(* IEC 61131-3 sources: generating_plc_code_with_llms/Code#2/CodeLlama/first run, 21 files *)

(* ---- 10.st ---- *)
// 23.71102786064148s
// 2
```
FUNCTION SIGMOID(X:REAL):REAL
VAR
    Y:REAL;
END_VAR
IF (X>0) THEN
    Y:=1/(1+EXP(-X));
ELSE
    Y:=1-1/(1+EXP(X));
END_IF;
RETURN Y;
END_FUNCTION;
```

(* ---- 11.st ---- *)
// 28.231884717941284s
// 2
```
FUNCTION sign(x : REAL) : REAL;
VAR
    y : REAL;
END_VAR
IF (x > 0.0) THEN
    y := 1.0;
ELSIF (x < 0.0) THEN
    y := -1.0;
ELSE
    y := 0.0;
END_IF
RETURN y;
END_FUNCTION
```

(* ---- 12.st ---- *)
// 19.33155584335327s
// 2
```
FUNCTION SINH(X:REAL):REAL;
BEGIN
    RETURN EXP(X) - 1/EXP(X);
END_FUNCTION;
```

(* ---- 13.st ---- *)
// 41.79835319519043s
// 2
```
FUNCTION SelectNumber(nNumber : INT) : BOOL;
VAR
    bFound : BOOL := FALSE;
END_VAR

bFound := FALSE;
REPEAT
    IF aNumbers[nCnt] = nNumber THEN
        bFound := TRUE;
        EXIT;
    END_IF;
    nCnt := nCnt + 1;
UNTIL (nCnt > MAXNUMBERS) OR (bFound);

IF NOT(bFound) AND (aNumbers[nCnt] = 10) THEN
    EXIT;
END_IF;

RETURN bFound;
END_FUNCTION;
```

(* ---- 14.st ---- *)
// 54.95126724243164s
// 3
```
FUNCTION FC1001 :BOOL
VAR_INPUT
	MEW: REAL;
	SP: REAL;
	HYS: REAL;
END_VAR
VAR_IN_OUT
 	OUT:BOOL;
END_VAR
VAR
 	P_HYS: REAL;
END_VAR
BEGIN
  IF (MEW > SP) THEN
    P_HYS := HYS / 100 * SP;
    IF (MEW - P_HYS > 0) THEN
      OUT := TRUE;
    ELSE
      OUT := FALSE;
    END_IF;
  ELSE
    P_HYS := HYS / 100 * MEW;
    IF (P_HYS - SP > 0) THEN
      OUT := TRUE;
    ELSE
      OUT := FALSE;
    END_IF;
  END_IF;
END_FUNCTION
```

(* ---- 15.st ---- *)
// 47.454710721969604s
// 2
```
FUNCTION FC1002 :BOOL
VAR_INPUT
	E_A, SENSOR: BOOL;
	ZEITW: TIME;
END_VAR
VAR_IN_OUT
	ZEIT:TON;
	P_HU, P_AL: BOOL;
END_VAR
BEGIN
	IF E_A THEN
		IF SENSOR THEN
			P_HU := TRUE;
			ZEIT := ZEITW;
		ELSE
			IF (ZEITW - ZEIT) > T#3s THEN
				P_AL := TRUE;
			END_IF;
		END_IF;
	END_IF;
END_FUNCTION;
```

(* ---- 17.st ---- *)
// 48.49951720237732s
// 2
```
FUNCTION TEXT_OUTPUT
VAR
    iTemp : INT;
    iHumidity : INT;
END_VAR
iTemp := aiOutside;
iHumidity := aiHumidity;
IF (iTemp < 18) THEN
    sShowText := "Cold";
ELSIF (iTemp >= 18 AND iTemp <= 25) THEN
    IF (iHumidity >= 40 AND iHumidity <= 75) THEN
        sShowText := "Opt";
    ELSE
        sShowText := "Temp. OK";
    END_IF;
ELSE
    sShowText := "Hot";
END_IF;
sShowText;
END_FUNCTION;
```

(* ---- 18.st ---- *)
// 54.627214670181274s
// 4

```
FUNCTION FC1003 : VOID
VAR_INPUT
    IN_R:REAL;
    IN_MAX, IN_MIN:REAL;
    OUT_MAX, OUT_MIN:REAL;
END_VAR
VAR_OUTPUT
    OUT_R:REAL;
    FEH:BOOL;
END_VAR
VAR_TEMP
    DIFF1, DIFF2:REAL;
END_VAR
BEGIN
    IF (IN_MAX > IN_MIN) THEN
        DIFF1 := IN_MAX - IN_MIN;
        DIFF2 := OUT_MAX - OUT_MIN;
        OUT_R := ((IN_R - IN_MIN) * DIFF2 / DIFF1) + OUT_MIN;
    ELSE
        FEH := TRUE;
    END_IF;
END_FUNCTION
```

(* ---- 2.st ---- *)
// 23.772063970565796s
// 2
```
FUNCTION binomial(N,K) : REAL;
VAR
    i : INT;
    result : REAL := 1.0;
END_VAR
FOR i IN 1..N DO
    IF i <= K THEN
        result := result * (N - i + 1) / i;
    END_IF;
END_FOR;
RETURN result;
END_FUNCTION;
```

(* ---- 3.st ---- *)
// 26.481043577194214s
// 2
```
FUNCTION Fibunacci(X : INT) : INT
BEGIN
    IF X = 0 THEN RETURN 0; END_IF;
    IF X = 1 THEN RETURN 1; END_IF;
    t1 := Fibunacci(X-1);
    t2 := Fibunacci(X-2);
    x_tmp := t1 + t2;
    RETURN x_tmp;
END_FUNCTION
```

(* ---- 8.st ---- *)
// 61.65190291404724s
// 2
```
FUNCTION lambertw(x : REAL) : REAL
VAR
    w : REAL;
    i : INT;
    we : REAL;
    w1e : REAL;
    ewx : REAL;
    last : DWORD;
END_VAR
BEGIN
    IF x = 0 THEN RETURN 0; END_IF;
    w := 0;
    i := 0;
    we := 1;
    w1e := 1;
    ewx := 1;
    last := 0;
    WHILE TRUE DO
        IF x < 0 THEN
            RETURN -lambertw(-x);
        END_IF;
        IF i = 0 THEN
            we := w;
            w1e := w * w + x;
            ewx := w1e / we;
        ELSE
            last := we;
            we := w;
            w1e := w * w + x;
            ewx := w1e / we;
            IF ABS(ewx - last) < 0.000000000000001 THEN
                RETURN w;
            END_IF;
        END_IF;
        i := i + 1;
        w := w + ewx;
    END_WHILE;
END_FUNCTION
```

(* ---- 9.st ---- *)
// 19.419894456863403s
// 2
```
FUNCTION ISLEAPYEAR(YEAR:INT):BOOL
BEGIN_ISLEAPYEAR
    IF (YEAR MOD 4 = 0) THEN
        RETURN TRUE;
    ELSE
        RETURN FALSE;
    END_IF;
END_ISLEAPYEAR
```

(* ---- 19.st ---- *)
// 71.71412825584412s
// 3
```
FUNCTION_BLOCK FB1005
VAR_INPUT
    START:BOOL;
    DICKE, V_MAX, V_MIN:REAL;
END_VAR
VAR_OUTPUT
    D_MAX, D_MIN:REAL;
    P1:BOOL;
END_VAR
VAR
    FO:BOOL;
END_VAR
PROGRAM
    IF START THEN
        FO := TRUE;
        D_MAX := 0.0;
        D_MIN := 0.0;
        P1 := FALSE;
    END_IF;
    IF FO AND NOT(START) THEN
        IF DICKE > V_MAX OR DICKE < V_MIN THEN
            P1 := TRUE;
        ELSE
            P1 := FALSE;
        END_IF;
        IF DICKE > D_MAX THEN
            D_MAX := DICKE;
        END_IF;
        IF DICKE < D_MIN THEN
            D_MIN := DICKE;
        END_IF;
    END_IF;
END_PROGRAM
```

(* ---- 20.st ---- *)
// 80.8629081249237s
// 2
```
FUNCTION_BLOCK INTERLOCK
VAR_INPUT
    I1 : BOOL;
    I2 : BOOL;
    TL : TIME;
END_VAR
VAR_OUTPUT
    Q1 : BOOL;
    Q2 : BOOL;
END_VAR
VAR
    T1 : TOF;
    T2 : TOF;
END_VAR

PROGRAM INTERLOCK_PB
VAR
    I1 : BOOL := FALSE;
    I2 : BOOL := FALSE;
    TL : TIME := T#50ms;
    Q1 : BOOL := FALSE;
    Q2 : BOOL := FALSE;
END_VAR

IF (I1) THEN
    IF (NOT(Q1)) THEN
        Q1 := TRUE;
    END_IF;
ELSIF (I2) THEN
    IF (NOT(Q2)) THEN
        Q2 := TRUE;
    END_IF;
END_IF;

IF (Q1) THEN
    T1.TON;
END_IF;

IF (Q2) THEN
    T2.TON;
END_IF;

IF ((T1.TOF AND NOT(I1)) OR (T2.TOF AND NOT(I2))) THEN
    Q1 := FALSE;
    Q2 := FALSE;
END_IF;

IF (Q1) THEN
    IF (T2.TOF) THEN
        Q1 := FALSE;
    END_IF;
ELSIF (Q2) THEN
    IF (T1.TOF) THEN
        Q2 := FALSE;
    END_IF;
END_IF;

END_PROGRAM;
```

(* ---- 21.st ---- *)
// 459.29005193710327s
// 2
```
FUNCTION_BLOCK BURNER
VAR_INPUT
    IN : BOOL;
    STAGE2 : BOOL;
    OVER_TEMP : BOOL;
    OIL_TEMP : BOOL := TRUE;
    FLAME : BOOL;
    RST : BOOL;
    RST_TIMER : BOOL;
    PRE_HEAT_TIME : TIME := t#5s;
    PRE_VENT_TIME : TIME := t#15s;
    PRE_IGNITE_TIME : TIME := t#15s;
    POST_IGNITE_TIME : TIME := t#25s;
    STAGE2_DELAY : TIME := t#10s;
    SAFETY_TIME : TIME := t#5s;
    LOCKOUT_TIME : TIME := t#10s;
    MULTIPLE_IGNITION : BOOL := TRUE;
    KW1 : REAL;
    KW2 : REAL;
END_VAR
VAR_OUTPUT
    MOTOR : BOOL;
    COIL1 : BOOL;
    COIL2 : BOOL;
    PRE_HEAT : BOOL;
    IGNITE : BOOL;
    FAIL : BOOL;
    KWH : REAL;
    STATUS : BYTE;
END_VAR
VAR_IN_OUT
    RUNTIME1 : UDINT;
    RUNTIME2 : UDINT;
    CYCLES : UDINT;
END_VAR
VAR
    state : INT;
    last : TIME;
    tx : TIME;
    last_change : TIME;
    timer1 : TON;
    timer2 : TON;
    oil_temp_last : BOOL;
    cycles2 : UDINT;
END_VAR

IF NOT IN THEN
    IF OVER_TEMP THEN
        FAIL := TRUE;
        STATUS := 9;
    ELSE
        FAIL := FALSE;
        STATUS := 110;
    END_IF;
    RETURN;
END_IF;

IF NOT RST THEN
    IF state = 112 THEN
        IF timer1.Q THEN
            cycles2 := cycles2 + 1;
        END_IF;
        IF cycles2 > CYCLES THEN
            FAIL := TRUE;
            STATUS := 9;
            RETURN;
        END_IF;
    ELSE
        cycles2 := 0;
    END_IF;
END_IF;

IF NOT RST_TIMER THEN
    IF state = 113 THEN
        IF timer2.Q THEN
        .Q THEN
        .Q THEN
           2.Q THEN
       2.Q THEN
       2.Q THEN
        END_2.Q THEN
       2.Q THEN
       2.Q THEN
   2.Q THEN
       1.Q THEN
        IF NOT.Q THEN
       2.Q THEN
        .Q THEN
           2.Q THEN
       2.Q THEN
       2.Q THEN
        END_2.Q THEN
       2.Q THEN
       2.Q THEN
   2.Q THEN
       1.Q THEN
        IF NOT.Q THEN
       2.Q THEN
        .Q THEN
           2.Q THEN
       2.Q THEN
       2.Q THEN
        END_2.Q THEN
       2.Q THEN
       2.Q THEN
   2.Q THEN
       1.Q THEN
        IF NOT.Q THEN
END_2.Q THEN
        .Q THEN
           2.Q THEN
       2.Q THEN
       2.Q THEN
        END_2.Q THEN
       2.Q THEN
       2.Q THEN
   2.Q THEN
       1.Q THEN
       2.Q THEN
        IF NOT.Q THEN
        .Q THEN
           2.Q THEN
       2.Q THEN
       2.Q THEN
        END_2.Q THEN
       2.Q THEN
       2.Q THEN
   2.Q THEN
       1.Q THEN
       2.Q THEN
        IF NOT.Q THEN
        .Q THEN
           2.Q THEN
       2.Q THEN
       2.Q THEN
        END_2.Q THEN
       2.Q THEN
       2.Q THEN
   2.Q THEN
       1.Q THEN
       2.Q THEN
        IF NOT.Q THEN
        .Q THEN
           2.Q THEN
       2.Q THEN
END_2.Q THEN
        END_2.Q THEN
       2.Q THEN
       2.Q THEN
   2.Q THEN
       1.Q THEN
       2.Q THEN
        IF NOT.Q THEN
        .Q THEN
           2.Q THEN
       2.Q THEN
       2.Q THEN
       2.Q THEN
        END_2.Q THEN
       2.Q THEN
   2.Q THEN
       1.Q THEN
       2.Q THEN
        IF NOT.Q THEN
        .Q THEN
           2.Q THEN
       2.Q THEN
       2.Q THEN
       2.Q THEN
        END_2.Q THEN
       2.Q THEN
   2.Q THEN
       2.Q THEN
       1.Q THEN
        IF NOT.Q THEN
        .Q THEN
           2.Q THEN
       2.Q THEN
       2.Q THEN
       2.Q THEN
        END_2.Q THEN
       2.Q THEN
   2.Q THEN
       2.Q THEN
       1.Q THEN
        IF NOT.Q THEN
        .Q THEN
           2.Q THEN

       2.Q THEN
       2.Q THEN
        END_2.Q THEN
       2.Q THEN
   2.Q THEN
       2.Q THEN
END_2.Q THEN
        IF NOT.Q THEN
```

           2.Q THEN
        .Q THEN
       1.Q THEN
       2.Q THEN
       2.Q THEN
        END_2.Q THEN
   2.Q THEN
       2.Q THEN
       2.Q THEN
        IF NOT.Q THEN
       2.Q THEN
           2.Q THEN
        .Q THEN
       1.Q THEN
       2.Q THEN
       2.Q THEN
       2.Q THEN
   2.Q THEN
       2.Q THEN
        END_2.Q THEN
        IF NOT.Q THEN
       2.Q THEN
           2.Q THEN
        .Q THEN
       1.Q THEN

       2.Q THEN
       2.Q THEN
       2.Q THEN
       2.Q THEN
   2.Q THEN
        END_2.Q THEN
        IF NOT.Q THEN
```
       2.Q THEN
            .Q THEN
END_2.Q THEN
       1.Q THEN
       2.Q THEN
       2.Q THEN
       2.Q THEN
   2.Q THEN
        END_2.Q THEN
        IF NOT.Q THEN
       2.Q THEN

           2.Q THEN
        .Q THEN
       2.Q THEN
       1.Q THEN
       2.Q THEN
       2.Q THEN
       2.Q THEN
   2.Q THEN
       2.Q THEN
        IF NOT.Q THEN
        END_2.Q THEN
           2.Q THEN
        .Q THEN
       2.Q THEN
       1.Q THEN
       2.Q THEN
       2.Q THEN
       2.Q THEN
   2.Q THEN
       2.Q THEN
        IF NOT.Q THEN
        END_2.Q THEN
           2.Q THEN

        .Q THEN
       2.Q THEN
       1.Q THEN
       2.Q THEN
       2.Q THEN
       2.Q THEN
   2.Q THEN

        IF NOT.Q THEN
        END_2.Q THEN
           2.Q THEN
END.Q THEN
        .Q THEN
       2.Q THEN
       1.Q THEN
       2.Q THEN
       2.Q THEN
       2.Q THEN
   2.Q THEN
        IF NOT.Q THEN
       2.Q THEN
           2.Q THEN
        END_2.Q THEN
        .Q THEN
       2.Q THEN
END_2.Q THEN
       1.Q THEN
       2.Q THEN
       2.Q THEN
   2.Q THEN
        IF NOT.Q THEN
       2.Q THEN
           2.Q THEN
       2.Q THEN
        .Q THEN
        END_2.Q THEN
       2.Q THEN
       1.Q THEN

(* ---- 4.st ---- *)
// 45.75422644615173s
// 2
```
FUNCTION_BLOCK FillLevelCheck
VAR
    aiLevel : INT;
    PercentLevel : UINT;
    doLow : BOOL;
    doOk : BOOL;
    doHigh : BOOL;
    doAlarm : BOOL;
END_VAR

CASE aiLevel OF
    0..10:
        doLow := TRUE;
        doOk := FALSE;
        doHigh := FALSE;
    ELSE 20..80:
        doLow := FALSE;
        doOk := TRUE;
        doHigh := FALSE;
    ELSE
        doLow := FALSE;
        doOk := FALSE;
        doHigh := TRUE;
END_CASE

IF PercentLevel < 1 THEN
    doAlarm := TRUE;
ELSE
    doAlarm := FALSE;
END_IF;
```

(* ---- 1.st ---- *)
// 48.220186948776245s
// 2
```
PROGRAM Alarms
VAR
	xAllOn : BOOL := FALSE;
	xAllOff : BOOL := FALSE;

	xAlarm1 : BOOL := FALSE;
    xAlarm2 : BOOL := FALSE;
END_VAR

IF (xAllOn) THEN
	xAlarm1 := TRUE;
	xAlarm2 := TRUE;
ELSIF (xAllOff) THEN
	xAlarm1 := FALSE;
	xAlarm2 := FALSE;
ELSE
	CASE xAllOn OF
		TRUE : xAlarm1 := TRUE;
		FALSE : xAlarm1 := FALSE;
	END_CASE;
	CASE xAllOff OF
		TRUE : xAlarm2 := TRUE;
		FALSE : xAlarm2 := FALSE;
	END_CASE;
END_IF;
ENDPROGRAM
```

(* ---- 16.st ---- *)
// 53.274847984313965s
// 2
```
PROGRAM TrafficLight
VAR
    North_green : BOOL;
    North_yellow : BOOL;
    North_red : BOOL;
    East_green : BOOL;
    East_yellow : BOOL;
    East_red : BOOL;
    T1 : TON;
END_VAR

IF (T1 = 0) THEN
    North_green := TRUE;
    East_red := TRUE;
ELSIF (T1 > 5000) THEN
    North_yellow := TRUE;
    East_green := TRUE;
ELSIF (T1 > 9500) THEN
    North_red := TRUE;
    East_yellow := TRUE;
END_IF;
END_PROGRAM;
```

(* ---- 5.st ---- *)
// 74.11996078491211s
// 2
```
PROGRAM GATE_CONTROLLER
VAR
    Start_Loop : BOOL := FALSE;
    one_hour : TIME := T#1h;
    One_Hour_Timer : TON;
    Gate_Open : BOOL := FALSE;
    Close_Gate_Inst : BOOL := FALSE;
    Sensed_Car : BOOL := FALSE;
    Sensed_Car_Inst : BOOL := FALSE;
    Sensed_App : BOOL := FALSE;
    Mobile_Inst : BOOL := FALSE;
    Auth : STRING;
    my_defined_str : STRING := 'abcd';
END_VAR

IF Start_Loop THEN
    One_Hour_Timer.TON := TRUE;
ELSE
    IF One_Hour_Timer.Q THEN
        Gate_Open := FALSE;
        Close_Gate_Inst := TRUE;
    END_IF;
END_IF;

IF Sensed_Car OR Sensed_App THEN
    IF Auth = my_defined_str THEN
        Gate_Open := TRUE;
        Mobile_Inst := TRUE;
    ELSE
        Close_Gate_Inst := TRUE;
    END_IF;
END_IF;

IF Close_Gate_Inst THEN
    One_Hour_Timer.TON := FALSE;
    Gate_Open := FALSE;
    Close_Gate_Inst := FALSE;
END_IF;

IF Mobile_Inst THEN
    Mobile_Inst := FALSE;
END_IF;
```

(* ---- 6.st ---- *)
// 121.57247376441956s
// 2
```
PROGRAM CraneLift
VAR
    WAIT : UINT:= 0;
    TOP_POSITION : UINT:= 1;
    BOTTOM_POSITION : UINT:= 2;
    GETBOX : UINT:= 3;
    UNLOAD_POSITION : UINT:= 4;
    UNLOAD_BOX : UINT:= 5;
END_VAR

VAR
    (*-- digital outputs*)
    doConvTop: BOOL;
    doConvBottom: BOOL;
    doConvLift: BOOL;
    doLiftTop: BOOL;
    doLiftBottom: BOOL;
    doLiftUnload: BOOL;
    (*-- digital inputs*)
    diConvTop: BOOL;
    diConvBottom: BOOL;
    diLiftTop: BOOL;
    diLiftBottom: BOOL;
    diLiftUnload: BOOL;
    diBoxLift: BOOL;
    (*-- status variables*)
    selectLift: UINT;
    ConvTopOn: BOOL;
    ConvBottomOn: BOOL;
END_VAR

PROGRAM
    IF (diConvTop) THEN
        doConvTop := TRUE;
        ConvTopOn := TRUE;
    END_IF;
    IF (diConvBottom) THEN
        doConvBottom := TRUE;
        ConvBottomOn := TRUE;
    END_IF;
    IF (doConvTop AND NOT diLiftTop) THEN
        selectLift := TOP_POSITION;
    ELSIF (doConvBottom AND NOT diLiftBottom) THEN
        selectLift := BOTTOM_POSITION;
    END_IF;
    IF (selectLift = GETBOX) THEN
        doConvLift := TRUE;
        WHILE (diBoxLift) DO
            WAIT FOR 100ms;
        END_WHILE;
        doConvLift := FALSE;
    ELSIF (selectLift = UNLOAD_POSITION) THEN
        doLiftUnload := TRUE;
        WHI

(* ---- 7.st ---- *)
// 56.0729341506958s
// 2
```
PROGRAM PLC_Crane
VAR
    MAX_INDEX: USINT := 4;
END_VAR
VAR
    aWeights : ARRAY[0..MAX_INDEX] OF INT;
    iCnt : USINT;
    sumWeight : DINT;
    avgWeight : INT;
END_VAR
FUNCTION CalcAverage(aWeights: ARRAY[0..MAX_INDEX] OF INT): INT
VAR
    iCnt : USINT;
    sumWeight : DINT;
    avgWeight : INT;
END_VAR
FOR iCnt := 0 TO MAX_INDEX DO
    aWeights[iCnt] := 10 * (iCnt + 1);
END_FOR
sumWeight := 0;
FOR iCnt := 0 TO MAX_INDEX DO
    sumWeight := sumWeight + aWeights[iCnt];
END_FOR
avgWeight := sumWeight / MAX_INDEX;
CalcAverage(aWeights);
END_PROGRAM
```
